// Block: PrjConfig_A04

DATA_BLOCK PrjConfig_A04
VERSION : 0.1
   NON_RETAIN
   VAR
      Area04_Main : AreaConfig;
      A0303 : Struct
         Spalla : Struct
            Testa : Struct
               Ax : Positioning_DOL_Machine_Config;
               DelayMissingCondition : Time;
            END_STRUCT;
            Coda : Struct
               Ax : Positioning_DOL_Machine_Config;
               DelayMissingCondition : Time;
            END_STRUCT;
         END_STRUCT;
         Spintore : Struct
            Testa : Struct
               Vrt : ValveMachine_Config;
               Orz : ValveMachine_Config;
            END_STRUCT;
            Coda : Struct
               Vrt : ValveMachine_Config;
               Orz : ValveMachine_Config;
            END_STRUCT;
            DelayMissingCondition : Time;
         END_STRUCT;
         TraslazioneStrato : Struct
            Testa : Struct
               Ax : Positioning_EPOS_Machine_Config_NEW;
               Manip_Sostegno : ValveMachine_Config;
               Manip_Pareggiatore : ValveMachine_Config;
               SostegnoVrt : ValveMachine_Config;
            END_STRUCT;
            Coda : Struct
               Ax : Positioning_EPOS_Machine_Config_NEW;
               Manip_Sostegno : ValveMachine_Config;
               Manip_Pareggiatore : ValveMachine_Config;
               SostegnoVrt : ValveMachine_Config;
               DelayMissingCondition : Time;
            END_STRUCT;
            DelayMissingCondition : Time;
         END_STRUCT;
         Sollevamento : Struct
            Testa : Struct
               Ax : Positioning_DOL_Machine_Config;
            END_STRUCT;
            Coda : Struct
               Ax : Positioning_DOL_Machine_Config;
            END_STRUCT;
            DelayMissingCondition : Time;
         END_STRUCT;
         Sostegno : Struct
            Testa : Struct
               Ax : Positioning_DOL_Machine_Config;
               V_1 : ValveMachine_Config;
               V_2 : ValveMachine_Config;
               DelayMissingCondition : Time;
            END_STRUCT;
            Coda : Struct
               Ax : Positioning_DOL_Machine_Config;
               V_1 : ValveMachine_Config;
               V_2 : ValveMachine_Config;
               DelayMissingCondition : Time;
            END_STRUCT;
         END_STRUCT;
      END_STRUCT;
      A0304 : Struct
         Navetta : Struct
            Testa : Struct
               Ax : Positioning_DOL_Machine_Config;
               PalettiEsterni : ValveMachine_Config;
               PalettiInterni : ValveMachine_Config;
            END_STRUCT;
            Coda : Struct
               Ax : Positioning_DOL_Machine_Config;
               PalettiEsterni : ValveMachine_Config;
               PalettiInterni : ValveMachine_Config;
            END_STRUCT;
            DelayMissingCondition : Time;
         END_STRUCT;
      END_STRUCT;
   END_VAR

BEGIN
   // No initialization required
END_DATA_BLOCK
